PROGRAM Gate_Back_Move
VAR
	
	backGateGearIn		:MC_GearInDyn;
	backGateLeftAxisJog :MC_Jog;
	
END_VAR

(* 后龙门比较特殊，不是和大小龙门结构不一样，GearRatio需要测试*)

backGateGearIn(
	Master:= axis_BackGate_Left, 
	Slave:= axis_BackGate_Right, 
	Enable:= TRUE, 
	GearRatio:= 1, 
	Acceleration:= , 
	Deceleration:= , 
	Jerk:= , 
	BufferMode:= , 
	Options:= , 
	InGear=> , 
	Busy=> , 
	Active=> , 
	CommandAborted=> , 
	Error=> , 
	ErrorID=> );
	
	
backGateLeftAxisJog(
	Axis:= axis_BackGate_Left, 
	JogForward:= bBackGate_Up, 
	JogBackwards:= bBackGate_Down, 
	Mode:= , 
	Position:= , 
	Velocity:= , 
	Acceleration:= , 
	Deceleration:= , 
	Jerk:= , 
	Done=> , 
	Busy=> , 
	Active=> , 
	CommandAborted=> , 
	Error=> , 
	ErrorID=> );

END_PROGRAM

(* stored: Version 1.1.0.1, ProductVersion 3.1.4024.14
   POU Gate_Back_Move: Id {6b3b82ea-fe62-454c-a819-06a725bf7083}, SpecialFunc None *)
